TEXTLIST TL_E_MOVER_SELECTOR
  0 = 'SELECT_MOVER_INDEX'
  ! = 'SELECT_MOVER_AXIS_ID'
   = ''
END_TEXTLIST

(* stored: Version 1.1.0.1, ProductVersion 3.1.4026.13
   TextList TL_E_MOVER_SELECTOR: Id {2118ae42-00c6-4db1-8882-3f6f7783cc38} *)
